{attribute 'enable_dynamic_creation'}
FUNCTION_BLOCK FB_DBTransactionHandler
VAR_INPUT
	ProjectDBDefs : IProjectDBDefs; //Instance of the custom database FB for this database
END_VAR
VAR_OUTPUT
END_VAR
VAR
	//Property backing variables
	_JRSQLNetId : T_AmsNetID;
	_JRSQLPort : T_AmsPort;
	_DBServer : POINTER TO fb_dbserver;
	_Busy : BOOL;
	_Done : BOOL;
	_Error : BOOL;
	_ErrorId : UINT;	
	_ErrorText : STRING;
	
	//'Framework'
	bFirstScan: BOOL := TRUE;
	tmrState:  TON;

	nState:	UDINT	:= 0;
	nNextState:	UDINT	:= 0;
	bFirstEntry: BOOL;	
	
	//Locals
	Triggered : BOOL := FALSE;
	DataReturn : BOOL := FALSE;
	
	spName :STRING;
	spData: pvoid;
	spDataSize:UDINT;
	
	spDefinition : DBSPDefinition;
	spCallResult : DBSPCallResult;
	
	TransmitBuffer : POINTER TO BYTE;
	TransmitSize : UINT;
	ReceiveBuffer : POINTER TO BYTE;
	ReceiveSize : UINT;
	
	LastProcessTime : TIME;
		
	fbADSReadWrite: ADSRDWRTEX;

END_VAR
VAR CONSTANT
	cJRSQLTimeout : TIME := T#10S;
	cJRSQLCommandExecute : UDINT := 16#1000;
END_VAR

IF bFirstScan THEN
	nNextState:=0;
	nState:=9999;
	
	fbADSReadWrite(NETID:=_JRSQLNetId,PORT:=_JRSQLPort,WRTRD:=FALSE,TMOUT:=cJRSQLTimeout);
	bFirstScan := FALSE;
END_IF

//state machine	
IF nState <> nNextState THEN
	bFirstEntry := TRUE;
	nState := nNextState;
ELSE
	bFirstEntry := FALSE;
END_IF

tmrState(IN:=(NOT bFirstEntry), PT:=T#20S);

CASE nState OF
0:
	IF bFirstEntry THEN
		_Error:=FALSE;
		_ErrorId := 16#0;
		_ErrorText := '';
		_Done:=FALSE;
	END_IF

	IF Triggered THEN
		IF _DBServer^.Connected THEN
			nNextState := 40;
		ELSE
			nNextState := 10;
		END_IF
	END_IF
	
10://wait for connection
	IF (_DBServer^.Connected) THEN
		nNextState := 0;
	ELSIF tmrState.ET > cJRSQLTimeout THEN
		_ErrorText:='JRSQL connection timeout';		
		_ErrorId := 16#1;
		_Error:=TRUE;
		nNextState	:= 999;
 	END_IF

//States combined to get rid of scan delays	
40: //Call JRSQL
	IF bFirstEntry THEN
		IF(ProjectDBDefs.GetSPDef(spName, ADR(spDefinition))) THEN
			TransmitSize := SIZEOF(DBSPDefinition) + spDefinition.InputParamSize;
			ReceiveSize := SIZEOF(DBSPCallResult) + spDefinition.OutputParamSize;

			IF (spDataSize = spDefinition.InputParamSize+spDefinition.OutputParamSize) THEN
				;
			ELSE
				_ErrorText := CONCAT('Procedure data size mismatch. Expected: ',CONCAT(UINT_TO_STRING(spDefinition.InputParamSize+spDefinition.OutputParamSize),CONCAT(' Got: ',UDINT_TO_STRING(spDataSize))));
				_ErrorId:= 16#3;
				_Error:=TRUE;
				nNextState := 999;
			END_IF
		ELSE 
			_ErrorText:='Stored procedure not found';		
			_ErrorId := 16#2;
			_Error:=TRUE;
			nNextState	:= 999;		
		END_IF	
	
		IF (NOT _Error) THEN
			//Allocate buffers
			TransmitSize := SIZEOF(DBSPDefinition) + spDefinition.InputParamSize;
			TransmitBuffer := __NEW(BYTE, TransmitSize);
			MEMSET(TransmitBuffer,0,TransmitSize);
			ReceiveSize := SIZEOF(DBSPCallResult) + spDefinition.OutputParamSize;
			ReceiveBuffer := __NEW(BYTE, ReceiveSize);
			MEMSET(ReceiveBuffer,0,ReceiveSize);
		
			memcpy(TransmitBuffer,ADR(spDefinition),SIZEOF(DBSPDefinition));
			memcpy((TransmitBuffer + SIZEOF(DBSPDefinition)),spData,spDefinition.InputParamSize);
		END_IF
	END_IF

	IF (NOT _Error) THEN
		
		fbADSReadWrite(WRTRD:=TRUE, IDXGRP:=cJRSQLCommandExecute, WRITELEN:=TransmitSize, SRCADDR:= TransmitBuffer, READLEN:=ReceiveSize, DESTADDR:= ReceiveBuffer);

		IF NOT fbADSReadWrite.Busy THEN
			IF NOT fbADSReadWrite.ERR THEN
				memcpy(ADR(spCallResult),ReceiveBuffer,SIZEOF(DBSPCallResult));
			
				IF spCallResult.Result <> 1 THEN
					//Error returned by JRSQL
					_ErrorText := CONCAT('JRSQL error: ',spCallResult.ResultString);
					_ErrorId:= 16#1000 + spCallResult.Result;
					_Error:=TRUE;
					nNextState := 999;
				ELSE
					//Copy result to caller
					memcpy(spData+spDefinition.InputParamSize,ReceiveBuffer+SIZEOF(DBSPCallResult),spDefinition.OutputParamSize);
					LastProcessTime := spCallResult.ProcessTime;
					_Done:=TRUE;
					nNextState := 999;		
				END_IF
			ELSE
				IF fbADSReadWrite.ERRID = 1861 THEN
					_ErrorText := 'JRSQL response timeout';
					_ErrorId:= 16#8;
					_Error:=TRUE;
					nNextState := 999;	
				ELSE
					_ErrorText := Concat('Error communicating to JRSQL: ', UDINT_TO_STRING(fbADSReadWrite.ERRID));
					_ErrorId:= 16#9;
					_Error:=TRUE;
					nNextState := 999;	
				END_IF
			END_IF
		END_IF
	
		IF (nState <> nNextState) THEN
			fbADSReadWrite(WRTRD:=FALSE);
			__DELETE(TransmitBuffer);
			__DELETE(ReceiveBuffer);
		END_IF
	
	END_IF
	
999:
	IF bFirstEntry THEN
		IF NOT _Error THEN
			_Done:=TRUE;
		END_IF
	END_IF
	
	IF NOT Triggered THEN
		nNextState	:= 0;	
	END_IF

END_CASE	

_Busy := (nState <> 0);
Triggered:=FALSE;
DataReturn:=FALSE;

PROPERTY Busy : bool
GET
Busy := _Busy;
END_GET
END_PROPERTY

PROPERTY Done : bool
GET
Done := _Done;
END_GET
END_PROPERTY

PROPERTY Error : bool
GET
Error := _Error;
END_GET
END_PROPERTY

PROPERTY ErrorId : UDINT
GET
ErrorId := _ErrorId;
END_GET
END_PROPERTY

PROPERTY ErrorText : STRING
GET
ErrorText := _ErrorText;
END_GET
END_PROPERTY

METHOD ExecuteSP : BOOL
VAR_INPUT
	bForeground : BOOL;
	sSPName : STRING;
	pData : pvoid;
	nDataSize : UDINT;
END_VAR
VAR
	BackgroundItem : POINTER TO DBBackgroundItem;
	
	
END_VAR
IF bForeground THEN
	//execute in process
	IF NOT busy THEN
		//first time call, set data
		spName := sSPName;
		spData := pData;
		spDataSize := nDataSize;
	ELSE
		//subsequent call
	
	END_IF

	Triggered:=TRUE;
	DataReturn:=FALSE;
	ExecuteSP:=(_Done OR _Error);
ELSE
	//build a new item to disassociate from the caller
	BackgroundItem:= __NEW(DBBackgroundItem);
	BackgroundItem^.SPName := sSPName;
	BackgroundItem^.DataSize := nDataSize;
	memcpy(ADR(BackgroundItem^.Data),pData,nDataSize);
	
	//Pass it off to the background fifo	
	IF NOT (_DBServer^.AddBackgroundItem(BackgroundItem)) THEN
		//add failed, clear the memory

		__DELETE(BackgroundItem);
	END_IF
	
	ExecuteSP:=TRUE;
END_IF
END_METHOD

METHOD FB_init : BOOL
VAR_INPUT
	bInitRetains : BOOL; // if TRUE, the retain variables are initialized (warm start / cold start)
	bInCopyCode : BOOL;  // if TRUE, the instance afterwards gets moved into the copy code (online change)
	
	pDBServer : POINTER TO FB_DBServer; //Instance of the custom database FB for this database
	JRSQLNetId : T_AmsNetID := ''; //AMS address of JRSQL
	JRSQLPort : T_AmsPort := 2020; //AMS port of JRSQL
	ProjectDBDefs : IProjectDBDefs; //Project database config
	
END_VAR
_DBServer := pDBServer;
_JRSQLNetId := JRSQLNetId;
_JRSQLPort := JRSQLPort;
THIS^.ProjectDBDefs := ProjectDBDefs;

IF bInitRetains THEN
	bFirstScan := TRUE;
END_IF
END_METHOD

END_FUNCTION_BLOCK

(* stored: Version 1.1.0.1, ProductVersion 3.1.4024.6
   POU FB_DBTransactionHandler: Id {d6ededa3-61b3-4fa6-bf15-9e07ceeccb43}, SpecialFunc None
   Property Busy: Id {c5c3e301-7de1-4df5-8848-3563b4764913}
   Get Get: Id {7ad243eb-6c9f-4a9b-bd5c-841d508ed439}
   Property Done: Id {2d421aed-3ff2-403a-9fbd-1eb4e4d6b46b}
   Get Get: Id {f1da60f8-dd41-4104-a349-29c35405b4ab}
   Property Error: Id {f210fa07-4dfd-41cf-bd61-be643e481aaf}
   Get Get: Id {532ed6d2-950d-41b6-b900-cd4db1274848}
   Property ErrorId: Id {11d44da4-7138-45e8-937b-c29719888bf5}
   Get Get: Id {51efcc06-d768-4f74-a442-2e8631e33353}
   Property ErrorText: Id {3dc0884a-8fc7-4936-b842-35c840e4b93e}
   Get Get: Id {6a22ddf5-e4f8-41df-a02f-588fd8ffdb09}
   Method ExecuteSP: Id {7429cab3-8ffe-498c-99ed-bdb55fca476a}
   Method FB_init: Id {787457e6-e363-4b57-b9b5-cdb9c7d872da} *)
